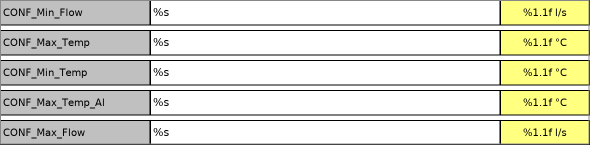
VISUALIZATION VISU_CONF_LIGNE_EAU_FLOWTEMP  // 590x145
VAR_IN_OUT
	m_Input_LIGNE_CONF_EAU : BLOCK_LIGNE_REF_FLOWTEMP;
END_VAR
    Rectangle (0,0 150x25), "CONF_Min_Flow"
    Rectangle (0,120 150x25), "CONF_Max_Flow", invisible if: true
    Rectangle (0,60 150x25), "CONF_Min_Temp"
    Rectangle (0,30 150x25), "CONF_Max_Temp"
    Rectangle (0,90 150x25), "CONF_Max_Temp_Al"
    Rectangle (500,0 90x25), "%1.1f l/s", text variable: m_Input_LIGNE_CONF_EAU.CONF_Min_Flow, input disabled if: NOT Global_Variables.PRG_USER.ACTU_USER.CONF_MACHINE OR m_Input_LIGNE_CONF_EAU.CONF_Max_Flow <= 0
        OnMouseClick: write the text variable via VisuDialogs.NumpadExtended, min 0, max m_Input_LIGNE_CONF_EAU.CONF_Max_Flow
    Rectangle (500,120 90x25), "%1.1f l/s", text variable: m_Input_LIGNE_CONF_EAU.CONF_Max_Flow, invisible if: true, input disabled if: NOT Global_Variables.PRG_USER.ACTU_USER.CONF_MACHINE
        OnMouseClick: write the text variable via VisuDialogs.NumpadExtended, min m_Input_LIGNE_CONF_EAU.CONF_Min_Flow, max 100
    Rectangle (500,60 90x25), "%1.1f °C", text variable: m_Input_LIGNE_CONF_EAU.CONF_Min_Temp, input disabled if: NOT Global_Variables.PRG_USER.ACTU_USER.CONF_MACHINE OR m_Input_LIGNE_CONF_EAU.CONF_Max_Temp <= 0
        OnMouseClick: write the text variable via VisuDialogs.NumpadExtended, min 0, max m_Input_LIGNE_CONF_EAU.CONF_Max_Temp
    Rectangle (500,30 90x25), "%1.1f °C", text variable: m_Input_LIGNE_CONF_EAU.CONF_Max_Temp, input disabled if: NOT Global_Variables.PRG_USER.ACTU_USER.CONF_MACHINE
        OnMouseClick: write the text variable via VisuDialogs.NumpadExtended, min m_Input_LIGNE_CONF_EAU.CONF_Min_Temp, max 100
    Rectangle (500,90 90x25), "%1.1f °C", text variable: m_Input_LIGNE_CONF_EAU.CONF_Max_Temp_AL, input disabled if: NOT Global_Variables.PRG_USER.ACTU_USER.CONF_MACHINE OR m_Input_LIGNE_CONF_EAU.CONF_Max_Temp <= 0
        OnMouseClick: write the text variable via VisuDialogs.NumpadExtended, min 0, max m_Input_LIGNE_CONF_EAU.CONF_Max_Temp
    Rectangle (150,0 350x25), "%s", text list: 'TextList_Servitudes', text index: 1
    Rectangle (150,120 350x25), "%s", invisible if: true, text list: 'TextList_Servitudes', text index: 2
    Rectangle (150,60 350x25), "%s", text list: 'TextList_Servitudes', text index: 3
    Rectangle (150,30 350x25), "%s", text list: 'TextList_Servitudes', text index: 4
    Rectangle (150,90 350x25), "%s", text list: 'TextList_Servitudes', text index: 5
END_VISUALIZATION

(* stored: Version 1.1.0.1, ProductVersion 3.1.4024.12
   Visu VISU_CONF_LIGNE_EAU_FLOWTEMP: Id {232274f4-91cc-4772-ab6d-cde7a00e2f6e} *)
